TYPE BuilderParameters :
STRUCT
	position : LREAL;
	distance : LREAL;
	velocity : LREAL;
	acceleration : LREAL;
	deceleration : LREAL;
	jerk : LREAL;
	buffer_mode : MotionBufferMode;
	ratio_numerator : LREAL;
	ratio_denominator : UINT;
END_STRUCT
END_TYPE

(* stored: Version 1.1.0.1
   DUT BuilderParameters: Id {548db3ec-1c7f-04ea-1b3a-f2ba0ddcf02f} *)
